Fanuc KAREL source: kc00013.KL

-- PROVISIONAL review KL for V1013-1; original PC SHA256 599d3f92032ff56d5b7e5abf50cd2273b05b8e86b13b457f51743765407c5457
-- Incomplete behavior may be omitted. Consult companion uncertainty JSON. Do not deploy.
PROGRAM KC00013
%NOLOCKGROUP
BEGIN
  -- UNRESOLVED_PC offsets 5-39; opcodes 27,22,22,22,22,22,31
  -- UNRESOLVED_PC offsets 44-48; opcodes 7F
END KC00013
